// TIA Portal V18 export
DATA_BLOCK "AHU_F_PID_Compact_RHT_regulator"   // DB173
// stored: AutoNumber false, DBAccessibleFromOPCUA true, InstanceOfName PID_Compact, OfSystemLibElement PID_Compact, OfSystemLibVersion 2.3
PID_Compact   // technology object, version 2.3
   // VAR_INPUT
   //    Setpoint : Real;
   //    Input : Real;
   //    Input_PER : Int;
   //    Disturbance : Real;
   //    ManualEnable : Bool;
   //    ManualValue : Real;
   //    ErrorAck : Bool;
   //    Reset : Bool;
   //    ModeActivate : Bool;
   // END_VAR
   // VAR_OUTPUT
   //    ScaledInput { ExternalWritable := 'False'} : Real;
   //    Output { ExternalWritable := 'False'} : Real;
   //    Output_PER { ExternalWritable := 'False'} : Int;
   //    Output_PWM { ExternalWritable := 'False'} : Bool;
   //    SetpointLimit_H { ExternalWritable := 'False'} : Bool;
   //    SetpointLimit_L { ExternalWritable := 'False'} : Bool;
   //    InputWarning_H { ExternalWritable := 'False'} : Bool;
   //    InputWarning_L { ExternalWritable := 'False'} : Bool;
   //    State { ExternalWritable := 'False'} : Int;
   //    Error { ExternalWritable := 'False'} : Bool;
   //    ErrorBits { ExternalWritable := 'False'} : DWord;
   // END_VAR
   // VAR_IN_OUT
   //    Mode : Int := 3;
   // END_VAR
   // VAR
   //    InternalDiagnostic : DWord;
   //    InternalVersion { ExternalWritable := 'False'} : DWord;
   //    InternalRTVersion : DWord;
   //    IntegralResetMode { S7_SetPoint := 'True'} : Int;
   //    OverwriteInitialOutputValue : Real;
   //    RunModeByStartup { S7_SetPoint := 'True'} : Bool;
   //    LoadBackUp : Bool;
   //    SetSubstituteOutput { S7_SetPoint := 'True'} : Bool;
   //    PhysicalUnit { ExternalWritable := 'False'; S7_SetPoint := 'True'} : Int;
   //    PhysicalQuantity { ExternalWritable := 'False'; S7_SetPoint := 'True'} : Int := 1;
   //    ActivateRecoverMode { S7_SetPoint := 'True'} : Bool;
   // END_VAR
   // VAR RETAIN
   //    Warning { ExternalWritable := 'False'} : DWord;
   //    WarningInternal { ExternalWritable := 'False'} : DWord;
   // END_VAR
   // VAR
   //    Progress { ExternalWritable := 'False'} : Real;
   //    CurrentSetpoint { ExternalWritable := 'False'} : Real;
   //    CancelTuningLevel { S7_SetPoint := 'True'} : Real;
   //    SubstituteOutput { S7_SetPoint := 'True'} : Real;
   //    Config { S7_SetPoint := 'True'} : PID_CompactConfig;
   //    CycleTime { S7_SetPoint := 'True'} : PID_CycleTime;
   //    CtrlParamsBackUp { S7_SetPoint := 'True'} : PID_CompactControlParams;
   //    PIDSelfTune { S7_SetPoint := 'True'} : PID_CompactSelfTune;
   //    PIDCtrl { S7_SetPoint := 'True'} : PID_CompactControl;
   // END_VAR
   // VAR RETAIN
   //    Retain { S7_SetPoint := 'True'} : PID_CompactRetain;
   // END_VAR
BEGIN
   Config.InputPerOn := FALSE;
   Config.InputLowerLimit := -50.0;
END_DATA_BLOCK
